{attribute 'qualified_only'}
{attribute 'strict'}
TYPE PushoverMessageType :
(
	Monospace := 0,
  Html
) INT;
END_TYPE

(* stored: Version 1.1.0.1, ProductVersion 3.1.4024.12
   DUT PushoverMessageType: Id {5dfa10c6-a1ae-41a2-9710-f71fa765b682} *)
